Yaskawa INFORM job: R1_W08,11(-70,-90)_KM-OK.JBI

/JOB
//NAME R1_W08,11(-70,-90)_KM-OK
///FOLDERNAME KRIS-SCIANA
//POS
///NPOS 80,80,0,3,0,0
///TOOL 0
///POSTYPE PULSE
///PULSE
C00000=80634,56524,26439,-33552,116027,48375
C00001=80628,58269,45036,-31008,107028,51169
C00002=78911,55316,44053,-31183,105606,50866
C00003=78212,54208,43755,-31252,105015,50747
C00004=78077,53876,44572,-31170,104384,50872
C00005=78212,54208,43755,-31252,105015,50747
C00006=75675,58994,46299,-31860,104831,49753
C00007=75090,60550,48062,-31915,104366,49647
C00008=75675,58994,46299,-31860,104831,49753
C00009=73415,47128,27098,-33303,108822,47587
C00010=73012,45246,24655,-33476,109116,47321
C00011=73415,47128,27098,-33303,108822,47587
C00012=74150,48191,27319,-33287,109454,47700
C00013=75960,51015,28077,-33247,110987,47988
C00014=75965,52987,13601,-36257,119226,45094
C00015=136517,51935,5119,-1923,104393,8731
C00016=87157,-5483,-28306,57450,115604,41571
C00017=87147,-5039,-11335,53427,109619,37333
C00018=88649,-5898,-8462,52940,107396,36805
C00019=89258,-6153,-7236,52774,106498,36599
C00020=87889,14537,19903,58993,114209,37793
C00021=88767,13530,18983,59246,113694,37990
C00022=87889,14537,19903,58993,114209,37793
C00023=87649,13613,19920,58714,114095,37532
C00024=87889,14537,19903,58993,114209,37793
C00025=105942,-62521,-63510,26568,80862,38232
C00026=105031,-65851,-62417,26893,79012,37461
C00027=105195,-64382,-61180,26864,78954,37510
C00028=105031,-65851,-62417,26893,79012,37461
C00029=105431,-67258,-67024,26678,80780,38021
C00030=107641,-43424,-69167,26047,92329,41409
C00031=143143,24328,-21242,-15658,96224,-11878
C00032=72204,74256,59569,-26405,111997,60927
C00033=70917,68999,55676,-26710,111311,60566
C00034=85864,57700,53549,-32032,120643,64746
C00035=55390,23910,30993,-35423,95120,59471
C00036=70563,68474,57156,-26581,110137,60710
C00037=70776,68944,56037,-26701,111041,60575
C00038=82327,65803,62898,-33102,117932,64007
C00039=47664,10536,-3000,-36566,96935,55258
C00040=66932,87982,79688,-30579,103155,62915
C00041=68273,94194,85253,-30231,103438,63379
C00042=67652,72456,53103,-19372,121960,51858
C00043=68730,81297,71878,-24437,120905,53913
C00044=55201,6836,-5546,-939,98227,43617
C00045=66315,67012,49556,-19800,121060,51456
C00046=65775,67263,51320,-19811,120027,51426
C00047=71102,14960,-9600,-14779,110431,54727
C00048=68991,63069,47524,-18483,120952,52622
C00049=70206,68275,51151,-18045,121645,53017
C00050=67306,51124,50401,-20344,101560,40970
C00051=87477,30209,35148,-22218,113002,46164
C00052=88288,2949,10464,-26364,98256,51824
C00053=65224,53044,56715,-20613,98319,40767
C00054=65298,47795,50229,-20686,99552,40580
C00055=82340,17559,26624,-13359,101268,45963
C00056=71908,43018,52479,-24041,92531,45521
C00057=73734,43279,49847,-23760,94663,45760
C00058=75710,44802,35372,-24197,104128,44564
C00059=131785,47166,14001,-6017,108119,46057
C00060=158927,32103,13676,68669,79329,67442
C00061=158908,36411,34815,70732,75312,62704
C00062=161041,36978,37858,71079,73298,62259
C00063=161785,37979,40054,71314,72501,61974
C00064=161197,36103,37872,71200,73031,62071
C00065=161616,38399,39420,71134,72825,62225
C00066=160091,52730,61830,72934,71713,59121
C00067=159331,51665,59666,72650,72481,59393
C00068=153527,56458,59991,71753,77181,59746
C00069=155097,66673,45520,46808,107874,-38774
C00070=160646,74114,58732,46422,101973,-38891
C00071=161426,73397,58645,46444,101345,-38803
C00072=160874,72062,56896,46460,101906,-38810
C00073=161157,75917,61015,46390,101370,-38929
C00074=160608,85724,81128,45274,96442,-41505
C00075=159778,86810,81631,45169,97042,-41627
C00076=157799,88241,81814,44919,98490,-41911
C00077=156482,94558,73923,46181,104945,-39526
C00078=167679,39598,-22082,19335,97230,-42029
C00079=144689,40558,-40632,18601,81152,-34817
BC00000=15,446554,628321
BC00001=15,446554,628321
BC00002=15,446554,628321
BC00003=15,446554,628321
BC00004=15,446554,628321
BC00005=15,446554,628321
BC00006=15,446554,628321
BC00007=15,446554,628321
BC00008=15,446554,628321
BC00009=15,446554,628321
BC00010=15,446554,628321
BC00011=15,446554,628321
BC00012=15,446554,628321
BC00013=15,446554,628321
BC00014=15,446554,628321
BC00015=161990,534397,590954
BC00016=74827,482105,688957
BC00017=74827,482105,688957
BC00018=74827,482105,688957
BC00019=74827,482105,688957
BC00020=74827,482105,688957
BC00021=74827,482105,688957
BC00022=74827,482105,688957
BC00023=74827,482105,688957
BC00024=74827,482105,688957
BC00025=74827,482105,688957
BC00026=74827,482105,688957
BC00027=74827,482105,688957
BC00028=74827,482105,688957
BC00029=74827,482105,688957
BC00030=74827,482105,688957
BC00031=161990,523399,590954
BC00032=18200,449093,666099
BC00033=18200,449093,666099
BC00034=64204,449092,666090
BC00035=4865,381918,793092
BC00036=18200,449093,666099
BC00037=18200,449093,666099
BC00038=77068,449092,666090
BC00039=13661,368749,666090
BC00040=18200,449093,666099
BC00041=18200,449093,666099
BC00042=26785,438920,638446
BC00043=26785,438920,638446
BC00044=33903,430655,752210
BC00045=26785,438920,638446
BC00046=26785,438920,638446
BC00047=39931,438920,638446
BC00048=26785,438920,638446
BC00049=26785,438920,638446
BC00050=7685,432003,792502
BC00051=68177,432003,792502
BC00052=64162,432003,792502
BC00053=7685,432003,792502
BC00054=7685,432003,792502
BC00055=64162,432003,792502
BC00056=7685,432003,792502
BC00057=7685,432003,792502
BC00058=7685,432003,792502
BC00059=125249,527223,669995
BC00060=278947,484298,652650
BC00061=278947,484298,652650
BC00062=278947,484298,652650
BC00063=278946,484300,652649
BC00064=278947,484298,652650
BC00065=278947,484298,652650
BC00066=278947,484298,652650
BC00067=278947,484298,652650
BC00068=278947,484298,652650
BC00069=259918,478232,570644
BC00070=259918,478232,570644
BC00071=259918,478233,570643
BC00072=259918,478232,570644
BC00073=259918,478232,570644
BC00074=259918,478232,570644
BC00075=259918,478232,570644
BC00076=259918,478232,570644
BC00077=259918,478232,570644
BC00078=259919,478233,570641
BC00079=239349,626664,575206
///POSTYPE BASE
///RECTAN
///RCONF 0,0,0,0,1,0,0,0,0,0,0,0,0,0,0,0,0,0,0,0,0,0,0,0
P00006=2.006,1.622,-0.565,0.0000,0.0000,0.0000
P00021=0.073,2.058,-0.109,0.0000,0.0000,0.0000
///RCONF 0,0,0,0,0,0,0,0,0,0,0,0,0,0,0,0,0,0,0,0,0,0,0,0
P00026=2.644,0.055,-2.583,0.0000,0.0000,0.0000
//INST
///DATE 2025/05/20 14:58
///ATTR SC,RW
///GROUP1 RB1,BS1
NOP
'r2_W08,11(-70,-90)
'Path S787 (for W8)
SFTOF
MOVJ C00000 BC00000 VJ=50.00
MOVJ C00001 BC00001 VJ=100.00
MOVL C00002 BC00002 V=100.0
MOVL C00003 BC00003 V=60.0
REFP 3 C00004 BC00004
CALL JOB:SEARCH-R1
SET P021 P006
SFTON P021
MOVL C00005 BC00005 V=60.0
MOVL C00006 BC00006 V=60.0
REFP 3 C00007 BC00007
CALL JOB:SEARCH-R1
SET P021 P006
SFTON P021
MOVL C00008 BC00008 V=60.0
MOVL C00009 BC00009 V=60.0
REFP 3 C00010 BC00010
CALL JOB:SEARCH-R1
SET P021 P006
SFTON P021
MOVL C00011 BC00011 V=60.0
MOVL C00012 BC00012 V=100.0
MOVL C00013 BC00013 V=100.0
MOVL C00014 BC00014 V=100.0
MOVJ C00015 BC00015 VJ=100.00
'Path S867
SFTOF
MOVJ C00016 BC00016 VJ=100.00
MOVJ C00017 BC00017 VJ=100.00
MOVL C00018 BC00018 V=250.0
MOVL C00019 BC00019 V=166.7
MOVL C00020 BC00020 V=133.3
REFP 3 C00021 BC00021
CALL JOB:SEARCH-R1
SET P026 P006
SFTON P026
MOVL C00022 BC00022 V=133.3
REFP 3 C00023 BC00023
CALL JOB:SEARCH-R1
SET P026 P006
SFTON P026
MOVL C00024 BC00024 V=166.7
MOVL C00025 BC00025 V=166.7
MOVL C00026 BC00026 V=166.7
REFP 3 C00027 BC00027
CALL JOB:SEARCH-R1
SET P026 P006
SFTON P026
MOVL C00028 BC00028 V=166.7
MOVL C00029 BC00029 V=500.0
MOVL C00030 BC00030 V=1000.0
MOVJ C00031 BC00031 VJ=100.00
'Path W5
SFTOF
SFTON P021
CALL JOB:COFNIJ_DRUT
MOVJ C00032 BC00032 VJ=100.00
MOVL C00033 BC00033 V=100.0
COMM MOVL C00034 BC00034 V=100.0 PL=0
MOVL C00035 BC00035 V=100.0 PL=0
REFP 1 C00036 BC00036
REFP 2 C00037 BC00037
MACRO1 MJ#(0) ARGF6
ARCON
COMM MOVL C00038 BC00038 V=8.3
MOVL C00039 BC00039 V=8.3
ARCOF
MOVL C00040 BC00040 V=100.0
MOVL C00041 BC00041 V=100.0
SFTOF
'Path W6
SFTOF
SFTON P021
MOVJ C00042 BC00042 VJ=100.00
MOVL C00043 BC00043 V=100.0
MOVL C00044 BC00044 V=100.0 PL=0
REFP 1 C00045 BC00045
REFP 2 C00046 BC00046
MACRO1 MJ#(0) ARGF6
ARCON
MOVL C00047 BC00047 V=8.3
ARCOF
MOVL C00048 BC00048 V=100.0
MOVL C00049 BC00049 V=100.0
SFTOF
'Path W7
SFTOF
SFTON P021
MOVJ C00050 BC00050 VJ=100.00
MOVL C00051 BC00051 V=100.0
MOVL C00052 BC00052 V=100.0 PL=0
REFP 1 C00053 BC00053
REFP 2 C00054 BC00054
MACRO1 MJ#(0) ARGF6
ARCON
MOVL C00055 BC00055 V=8.3
ARCOF
MOVL C00056 BC00056 V=100.0
MOVL C00057 BC00057 V=100.0
MOVL C00058 BC00058 V=100.0
SFTOF
MOVJ C00059 BC00059 VJ=100.00
'
'Path W8
SFTOF
SFTON P026
MOVJ C00060 BC00060 VJ=100.00
MOVJ C00061 BC00061 VJ=100.00
MOVL C00062 BC00062 V=100.0
MOVL C00063 BC00063 V=100.0 PL=0
REFP 1 C00064 BC00064
REFP 2 C00065 BC00065
MACRO1 MJ#(0) ARGF6
ARCON
MOVL C00066 BC00066 V=8.3
ARCOF
MOVL C00067 BC00067 V=250.0
MOVJ C00068 BC00068 VJ=100.00
SFTOF
'Path W868
SFTOF
SFTON P026
MOVJ C00069 BC00069 VJ=100.00
MOVL C00070 BC00070 V=166.7
MOVL C00071 BC00071 V=100.0 PL=0
REFP 1 C00072 BC00072
REFP 2 C00073 BC00073
MACRO1 MJ#(0) ARGF6
ARCON
MOVL C00074 BC00074 V=8.3
ARCOF
MOVL C00075 BC00075 V=100.0
MOVL C00076 BC00076 V=100.0
MOVL C00077 BC00077 V=100.0
SFTOF
MOVJ C00078 BC00078 VJ=100.00
MOVJ C00079 BC00079 VJ=100.00
END
